(* PLC project Blank Project, Blank Blank 1.0 *)
(* stored: creationDateTime 2016-05-18T21:14:07, modificationDateTime 2018-01-26T14:59:05 *)

PROGRAM My_Program
  VAR
    OnOff AT %QX0.0 : BOOL := 0;
    MaxGen AT %IW0 : INT := 400;
    CurrentGen AT %IW1 : INT := 300;
    ID AT %IW2 : INT := 3;
    TargetGen AT %QW0 : INT := 300;
  END_VAR
  VAR
    Delta : INT := 2;
    Increasing : BOOL := 0;
    Decreasing : BOOL := 0;
    Tick : BOOL := 0;
    Tick_Count : INT := 0;
    TON0 : TON;
  END_VAR
  VAR  (* added by the conversion: wires and edge detectors of the diagram *)
    _MOVE50_OUT : BOOL;
    _MOVE4_OUT : BOOL;
    _MOVE11_OUT : BOOL;
    R_TRIG1 : R_TRIG;
    _MOVE36_OUT : BOOL;
    R_TRIG2 : R_TRIG;
    R_TRIG3 : R_TRIG;
    _GT125_OUT : BOOL;
  END_VAR

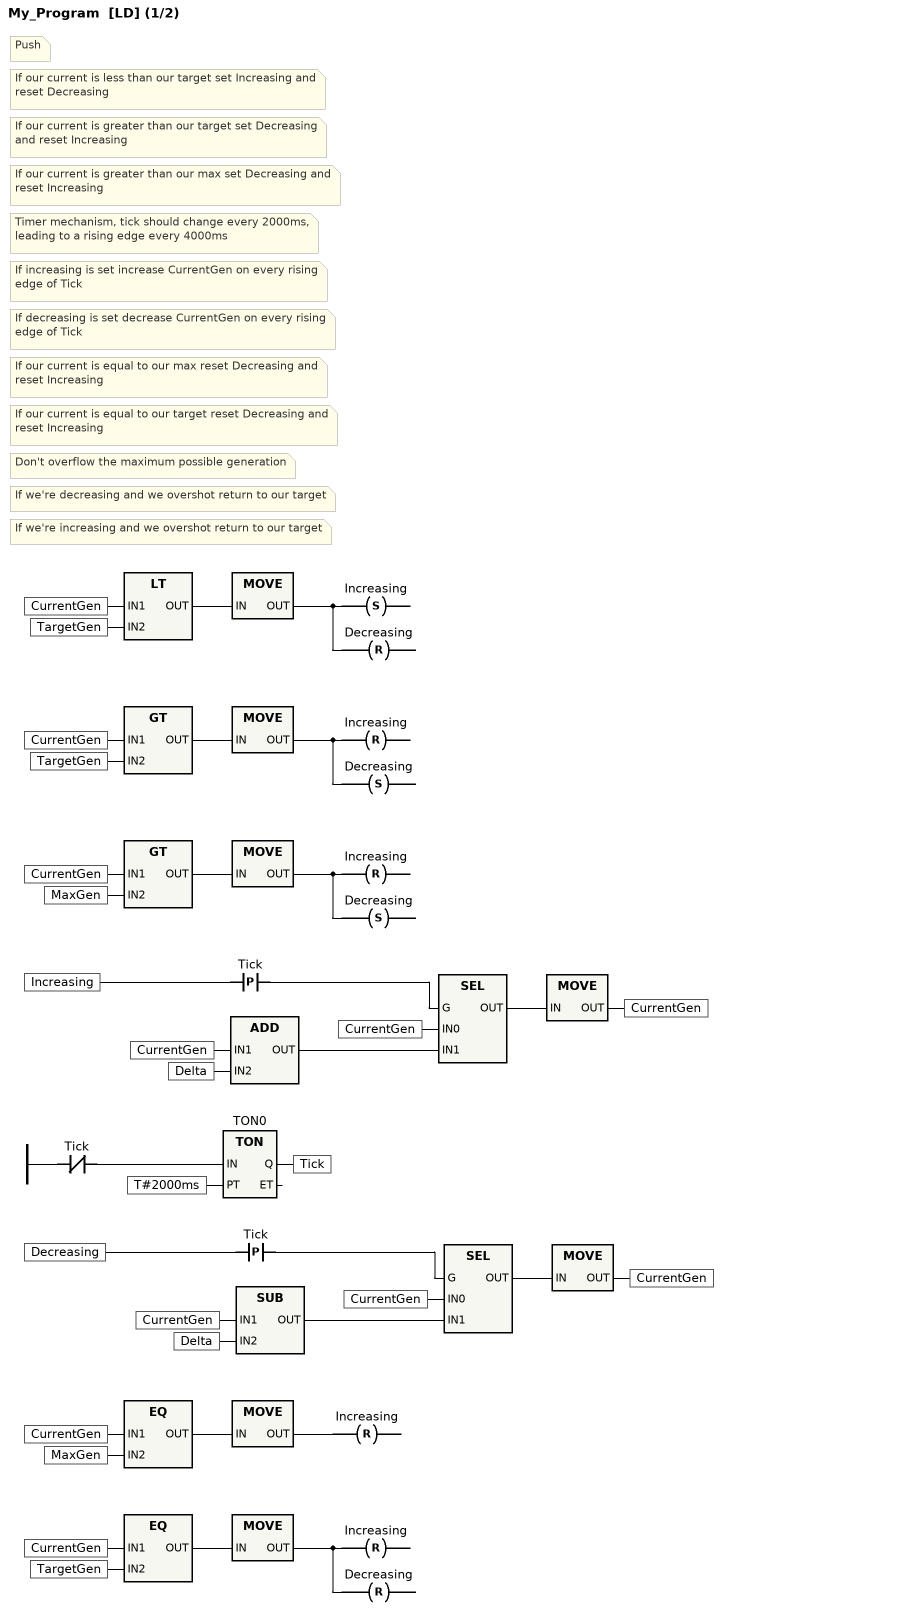
(* LD diagram, written out as Structured Text *)
_MOVE50_OUT := CurrentGen < TargetGen;
IF _MOVE50_OUT THEN Increasing := TRUE; END_IF;
(* If our current is less than our target set Increasing and reset Decreasing *)
IF _MOVE50_OUT THEN Decreasing := FALSE; END_IF;
_MOVE4_OUT := CurrentGen > TargetGen;
IF _MOVE4_OUT THEN Increasing := FALSE; END_IF;
(* If our current is greater than our target set Decreasing and reset Increasing *)
(* Timer mechanism, tick should change every 2000ms, leading to a rising edge every 4000ms *)
IF _MOVE4_OUT THEN Decreasing := TRUE; END_IF;
TON0(IN := NOT Tick, PT := T#2000ms);
Tick := TON0.Q;
_MOVE11_OUT := CurrentGen > MaxGen;
IF _MOVE11_OUT THEN Increasing := FALSE; END_IF;
(* If our current is greater than our max set Decreasing and reset Increasing *)
IF _MOVE11_OUT THEN Decreasing := TRUE; END_IF;
(* If our current is equal to our max reset Decreasing and reset Increasing *)
IF CurrentGen = MaxGen THEN Increasing := FALSE; END_IF;
R_TRIG1(CLK := Tick);
Tick_Count := SEL(1 AND R_TRIG1.Q, Tick_Count, 1 + Tick_Count);
_MOVE36_OUT := CurrentGen = TargetGen;
IF _MOVE36_OUT THEN Increasing := FALSE; END_IF;
(* If our current is equal to our target reset Decreasing and reset Increasing *)
IF _MOVE36_OUT THEN Decreasing := FALSE; END_IF;
R_TRIG2(CLK := Tick);
CurrentGen := SEL(Increasing AND R_TRIG2.Q, CurrentGen, CurrentGen + Delta);
(* If increasing is set increase CurrentGen on every rising edge of Tick *)
R_TRIG3(CLK := Tick);
CurrentGen := SEL(Decreasing AND R_TRIG3.Q, CurrentGen, CurrentGen - Delta);
(* If decreasing is set decrease CurrentGen on every rising edge of Tick *)
(* Don't overflow the maximum possible generation *)
TargetGen := MIN(TargetGen, MaxGen);
CurrentGen := MIN(CurrentGen, MaxGen);
(* If we're decreasing and we overshot return to our target *)
CurrentGen := SEL(TargetGen - CurrentGen > 0 AND TargetGen - CurrentGen < Delta AND Decreasing, CurrentGen, TargetGen);
(* If we're increasing and we overshot return to our target *)
CurrentGen := SEL(TargetGen - CurrentGen < 0 AND TargetGen - CurrentGen < Delta AND Increasing, CurrentGen, TargetGen);
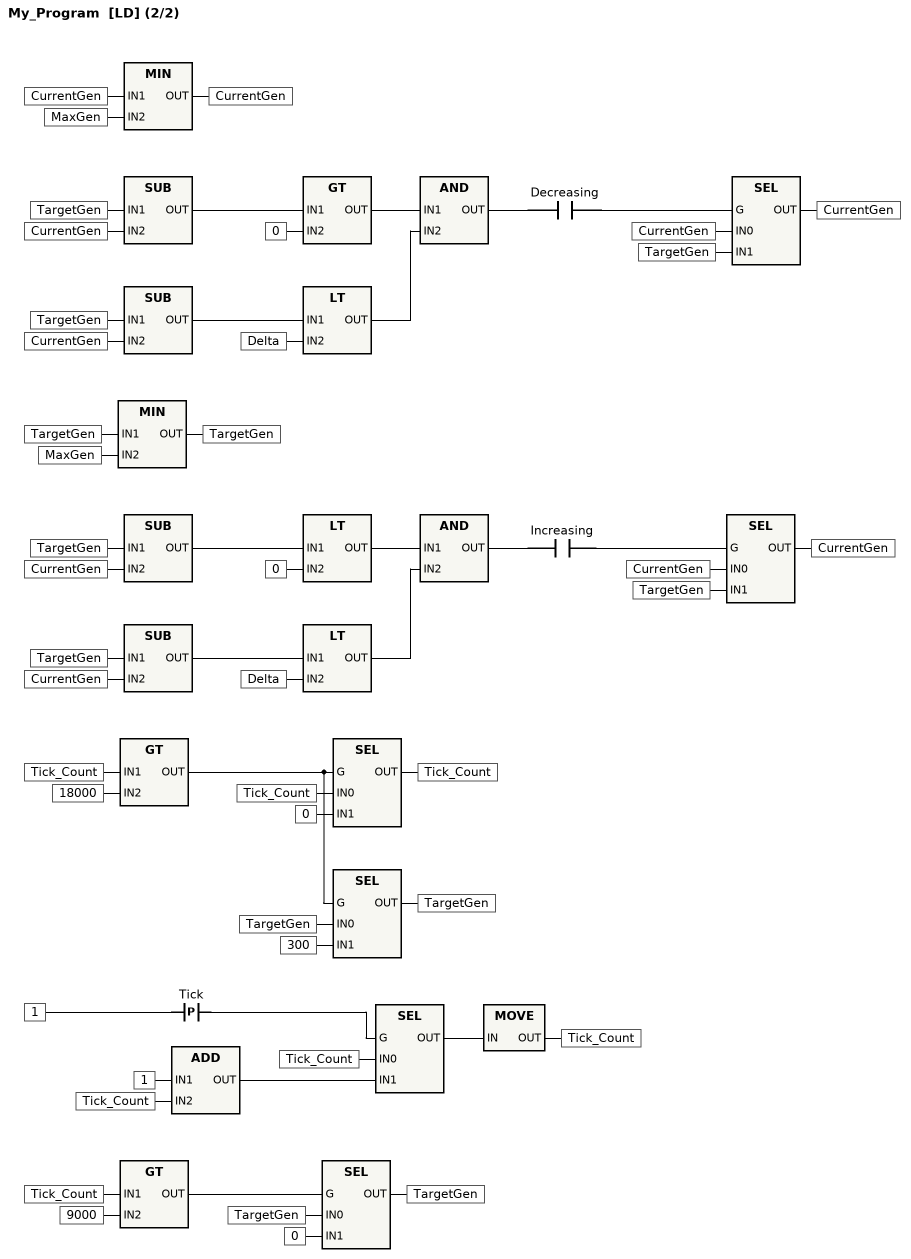
TargetGen := SEL(Tick_Count > 9000, TargetGen, 0);
_GT125_OUT := Tick_Count > 18000;
TargetGen := SEL(_GT125_OUT, TargetGen, 300);
Tick_Count := SEL(_GT125_OUT, Tick_Count, 0);
(* Push *)
END_PROGRAM

CONFIGURATION Config0
  RESOURCE Res0 ON PLC
    TASK TaskMain(INTERVAL := T#50ms, PRIORITY := 0);
    PROGRAM Inst0 WITH TaskMain : My_Program;
  END_RESOURCE
END_CONFIGURATION
